{attribute 'enable_dynamic_creation'}
FUNCTION_BLOCK FB_Helper
VAR
END_VAR

// Helper implementation

METHOD PUBLIC ImportConfigFromDB : BOOL
VAR_INPUT
	sFilePath : STRING(255);
END_VAR
// TODO: Implement file import
END_METHOD

METHOD PUBLIC LoadFrameConfigFromDB : BOOL
VAR_INPUT
	sFilePath : STRING(255);
END_VAR
// TODO: Implement frame config load
END_METHOD

METHOD PUBLIC LoadTargetConfigFromDB : BOOL
VAR_INPUT
	sFilePath : STRING(255);
END_VAR
// TODO: Implement target config load
END_METHOD

METHOD PUBLIC LoadToolConfigFromDB : BOOL
VAR_INPUT
	sFilePath : STRING(255);
END_VAR
// TODO: Implement tool config load
END_METHOD

METHOD PUBLIC SaveConfigToDB : BOOL
VAR_INPUT
	sFilePath : STRING(255);
END_VAR
// TODO: Implement file save
END_METHOD

METHOD PUBLIC SaveFrameConfigToDB : BOOL
VAR_INPUT
	sFilePath : STRING(255);
END_VAR
// TODO: Implement frame config save
END_METHOD

METHOD PUBLIC SaveTargetConfigToDB : BOOL
VAR_INPUT
	sFilePath : STRING(255);
END_VAR
// TODO: Implement target config save
END_METHOD

METHOD PUBLIC SaveToolConfigToDB : BOOL
VAR_INPUT
	sFilePath : STRING(255);
END_VAR
// TODO: Implement tool config save
END_METHOD

END_FUNCTION_BLOCK

(* stored: Version 1.1.0.1, ProductVersion 3.1.4026.18
   POU FB_Helper: Id {e1b2c3d4-1111-1111-1111-111111111111}, SpecialFunc None
   Method ImportConfigFromDB: Id {e1b2c3d4-1121-1111-1111-111111111111}
   Method LoadFrameConfigFromDB: Id {e1b2c3d4-1124-1111-1111-111111111111}
   Method LoadTargetConfigFromDB: Id {e1b2c3d4-1125-1111-1111-111111111111}
   Method LoadToolConfigFromDB: Id {e1b2c3d4-1123-1111-1111-111111111111}
   Method SaveConfigToDB: Id {e1b2c3d4-1122-1111-1111-111111111111}
   Method SaveFrameConfigToDB: Id {e1b2c3d4-1127-1111-1111-111111111111}
   Method SaveTargetConfigToDB: Id {e1b2c3d4-1128-1111-1111-111111111111}
   Method SaveToolConfigToDB: Id {e1b2c3d4-1126-1111-1111-111111111111} *)
